PROGRAM MAIN
VAR
	lineColor : E_LineColors;
END_VAR

PRG_DisconnectorExample();

PRG_ContactorExample();

PRG_CircuitBreakerExample();

PRG_Simulation();

PRG_LVCP1();

PRG_LVCP2();

PRG_LVCP5();

PRG_HVCP3();

PRG_HVCP5();

END_PROGRAM

(* stored: Version 1.1.0.1, ProductVersion 3.1.4024.14
   POU MAIN: Id {b4471795-9aa5-4506-a3bc-a219d6386ac6}, SpecialFunc None *)
